TYPE ST_HE_SATT_Status :
STRUCT
    bBusy : BOOL;
    bDone : BOOL;
    bError : BOOL;
    sErrorMsg : T_MaxString;
END_STRUCT
END_TYPE

(* stored: Version 1.1.0.1
   DUT ST_HE_SATT_Status: Id {ac4221c7-ab5c-421c-94c2-48698d888084} *)
